(*

.. <legal notes>

legal notes
=================
| SPDX-FileCopyrightText: © 2026 Oleksandr Tiutyk <trofimich@gmail.com>
| SPDX-License-Identifier: LGPL-3.0-only
| For details check: LGPL-3.0-only_

.. _LGPL-3.0-only: https://www.gnu.org/licenses/lgpl-3.0.en.html

.. </legal notes>

*)

PROGRAM SignedInt32Helper
VAR CONSTANT
	MIN_VALUE : DINT := -2_147_483_648;
	MAX_VALUE : DINT := +2_147_483_647;
	
	MIN_24BIT_VALUE : DINT := -8_388_608;
	MAX_24BIT_VALUE : DINT := +8_388_607;
END_VAR
VAR
	_ClassName : STRING := __POUNAME();
END_VAR

{attribute 'monitoring' := 'call'}
PROPERTY ClassName : STRING
GET
ClassName := _ClassName;
END_GET
END_PROPERTY

{attribute 'monitoring' := 'call'}
PROPERTY NamespaceName : STRING
GET
NamespaceName := CurrentNamespace.Name;
END_GET
END_PROPERTY

END_PROGRAM

(* stored: Version 1.1.0.1
   POU SignedInt32Helper: Id {36635b26-adca-4c25-86a1-647baaa97f3e}, SpecialFunc None
   Property ClassName: Id {9f4bff5c-648c-4bc4-8579-3a9863979e2d}
   Get Get: Id {3e65c282-f9dd-4064-a3e1-bc690a0ff61b}
   Property NamespaceName: Id {ed3fe1ed-9402-406f-86ad-dfa594726ef8}
   Get Get: Id {4a1470a8-ac41-4446-9b09-044a7d6d3de9} *)
